PROGRAM MAIN


//XTS Program Call
XTS_PRG();

END_PROGRAM

(* stored: Version 1.1.0.1, ProductVersion 3.1.4024.11
   POU MAIN: Id {85bca7ef-4594-424a-a11c-83d30e376864}, SpecialFunc None *)
